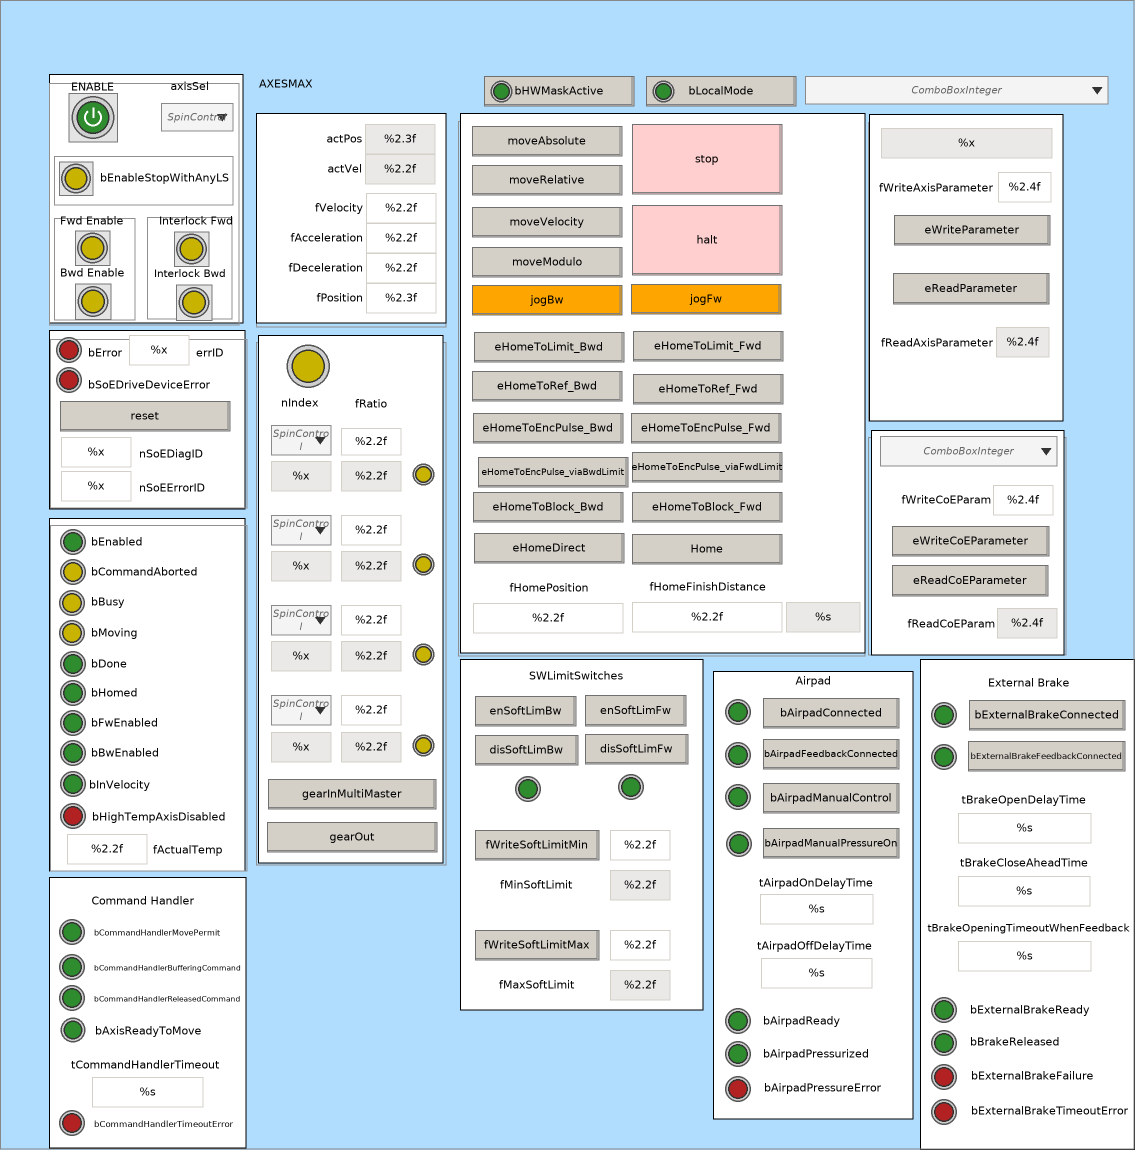
VISUALIZATION MainVisu  // 1135x1150
    Rectangle (49,518 196x353)
    Rectangle (49,330 196x179)
    Rectangle (49,877 197x271)
    Rectangle (49,74 194x249)
    GroupBox (868,114 195x307)
        Rectangle (1,0 194x307)
        Textfield (13,14 171x30), "%x", text variable: astAxes[MAIN.hmiAxisSelection].stConfig.eAxisParameters
            OnMouseClick: write GVL.astAxes[MAIN.hmiAxisSelection].stConfig.eAxisParameters via Default
        Textfield (130,58 53x30), "%2.4f", text variable: astAxes[MAIN.hmiAxisSelection].stConfig.fWriteAxisParameter
            OnMouseClick: write GVL.astAxes[MAIN.hmiAxisSelection].stConfig.fWriteAxisParameter via Default
        Button (26,101 156x30), "eWriteParameter", input disabled if: GVL.astAxes[MAIN.hmiAxisSelection].stStatus.bGeared, text list: "languageSupport", text index: "eWriteParameter"
            OnMouseClick: execute { GVL.astAxes[MAIN.hmiAxisSelection].stControl.eCommand:=E_MotionFunctions.eWriteParameter; GVL.astAxes[MAIN.hmiAxisSelection].stControl.bExecute:=TRUE; }
        Button (25,159 156x31), "eReadParameter", input disabled if: GVL.astAxes[MAIN.hmiAxisSelection].stStatus.bGeared, text list: 'languageSupport', text index: "eReadParameter"
            OnMouseClick: execute { GVL.astAxes[MAIN.hmiAxisSelection].stControl.eCommand:=E_MotionFunctions.eReadParameter; GVL.astAxes[MAIN.hmiAxisSelection].stControl.bExecute:=TRUE; }
        Textfield (128,213 53x30), "%2.4f", text variable: astAxes[MAIN.hmiAxisSelection].stConfig.fReadAxisParameter
            OnMouseClick: write GVL.astAxes[MAIN.hmiAxisSelection].stConfig.fReadAxisParameter via Default
    GroupBox (458,113 407x543)
        Rectangle (2,0 405x540)
        Button (174,92 150x70), "halt", pressed state: GVL.astAxes[Main.hmiAxisSelection].stControl.bHalt, input disabled if: GVL.astAxes[MAIN.hmiAxisSelection].stStatus.bGeared, text list: "languageSupport", text index: "halt"
            toggle GVL.astAxes[Main.hmiAxisSelection].stControl.bHalt
        Button (174,421 150x30), "Home", input disabled if: GVL.astAxes[MAIN.hmiAxisSelection].stStatus.bGeared, text list: 'languageSupport', text index: "Home"
            OnMouseClick: execute { GVL.astAxes[Main.hmiAxisSelection].stControl.eCommand:=E_MotionFunctions.eHome; GVL.astAxes[Main.hmiAxisSelection].stControl.bExecute:=TRUE; }
        Button (15,379 150x30), "eHomeToBlock_Bwd", input disabled if: GVL.astAxes[MAIN.hmiAxisSelection].stStatus.bGeared, text list: 'languageSupport', text index: "eHomeToBlock_Bwd"
            OnMouseClick: execute {
                GVL.astAxes[Main.hmiAxisSelection].stControl.eCommand:=E_MotionFunctions.eHome;
                GVL.astAxes[Main.hmiAxisSelection].stConfig.eHomeSeq:=E_HomingRoutines.eHomeToBlock_Bwd;
                GVL.astAxes[Main.hmiAxisSelection].stControl.bExecute:=TRUE;
            }
        Button (14,258 150x30), "eHomeToRef_Bwd", input disabled if: GVL.astAxes[MAIN.hmiAxisSelection].stStatus.bGeared, text list: 'languageSupport', text index: "eHomeToRef_Bwd"
            OnMouseClick: execute {
                GVL.astAxes[Main.hmiAxisSelection].stControl.eCommand:=E_MotionFunctions.eHome;
                GVL.astAxes[Main.hmiAxisSelection].stConfig.eHomeSeq:=E_HomingRoutines.eHomeToRef_Bwd;
                GVL.astAxes[Main.hmiAxisSelection].stControl.bExecute:=TRUE;
            }
        Button (14,13 150x30), "moveAbsolute", text list: "languageSupport", text index: "moveAbsolute"
            OnMouseClick: execute { GVL.astAxes[MAIN.hmiAxisSelection].stControl.eCommand:=E_MotionFunctions.eMoveAbsolute; GVL.astAxes[MAIN.hmiAxisSelection].stControl.bExecute:=TRUE; }
        Button (14,94 150x30), "moveVelocity", input disabled if: GVL.astAxes[MAIN.hmiAxisSelection].stStatus.bGeared, text list: "languageSupport", text index: "moveVelocity"
            OnMouseClick: execute { GVL.astAxes[Main.hmiAxisSelection].stControl.eCommand:=E_MotionFunctions.eMoveVelocity; GVL.astAxes[Main.hmiAxisSelection].stControl.bExecute:=TRUE; }
        Button (14,52 150x30), "moveRelative", input disabled if: GVL.astAxes[MAIN.hmiAxisSelection].stStatus.bGeared, text list: "languageSupport", text index: "moveRelative"
            OnMouseClick: execute { GVL.astAxes[Main.hmiAxisSelection].stControl.eCommand:=E_MotionFunctions.eMoveRelative; GVL.astAxes[Main.hmiAxisSelection].stControl.bExecute:=TRUE; }
        Button (14,134 150x30), "moveModulo", input disabled if: GVL.astAxes[MAIN.hmiAxisSelection].stStatus.bGeared, text list: "languageSupport", text index: "moveModulo"
            OnMouseClick: execute { GVL.astAxes[Main.hmiAxisSelection].stControl.eCommand:=E_MotionFunctions.eMoveModulo; GVL.astAxes[Main.hmiAxisSelection].stControl.bExecute:=TRUE; }
        Button (174,11 150x70), "stop", pressed state: GVL.astAxes[Main.hmiAxisSelection].stControl.bStop, input disabled if: GVL.astAxes[MAIN.hmiAxisSelection].stStatus.bGeared, text list: "languageSupport", text index: "stop"
            toggle GVL.astAxes[Main.hmiAxisSelection].stControl.bStop
        Button (14,172 150x30), "jogBw", text list: "languageSupport", text index: "jogBw"
            OnMouseDown: execute {
                GVL.astAxes[Main.hmiAxisSelection].stControl.eCommand:=E_MotionFunctions.eMoveVelocity;
                GVL.astAxes[Main.hmiAxisSelection].stControl.fVelocity:=-ABS(GVL.astAxes[Main.hmiAxisSelection].stControl.fJogVelocity);
                GVL.astAxes[Main.hmiAxisSelection].stControl.bExecute:= TRUE;
            }
            OnMouseUp: execute { GVL.astAxes[Main.hmiAxisSelection].stControl.bHalt:= TRUE; }
        Button (173,171 150x30), "jogFw", text list: "languageSupport", text index: "jogFw"
            OnMouseDown: execute {
                GVL.astAxes[Main.hmiAxisSelection].stControl.eCommand:=E_MotionFunctions.eMoveVelocity;
                GVL.astAxes[Main.hmiAxisSelection].stControl.fVelocity:=ABS(GVL.astAxes[Main.hmiAxisSelection].stControl.fJogVelocity);
                GVL.astAxes[Main.hmiAxisSelection].stControl.bExecute:= TRUE;
            }
            OnMouseUp: execute { GVL.astAxes[Main.hmiAxisSelection].stControl.bHalt:= TRUE; }
        Button (175,261 150x30), "eHomeToRef_Fwd", input disabled if: GVL.astAxes[MAIN.hmiAxisSelection].stStatus.bGeared, text list: "languageSupport", text index: "eHomeToRef_Fwd"
            OnMouseClick: execute {
                GVL.astAxes[Main.hmiAxisSelection].stControl.eCommand:=E_MotionFunctions.eHome;
                GVL.astAxes[Main.hmiAxisSelection].stConfig.eHomeSeq:=E_HomingRoutines.eHomeToRef_Fwd;
                GVL.astAxes[Main.hmiAxisSelection].stControl.bExecute:=TRUE;
            }
        Button (175,218 150x30), "eHomeToLimit_Fwd", input disabled if: GVL.astAxes[MAIN.hmiAxisSelection].stStatus.bGeared, text list: "languageSupport", text index: "eHomeToLimit_Fwd"
            OnMouseClick: execute {
                GVL.astAxes[Main.hmiAxisSelection].stControl.eCommand:=E_MotionFunctions.eHome;
                GVL.astAxes[Main.hmiAxisSelection].stConfig.eHomeSeq:=E_HomingRoutines.eHomeToLimit_Fwd;
                GVL.astAxes[Main.hmiAxisSelection].stControl.bExecute:=TRUE;
            }
        Button (16,219 150x30), "eHomeToLimit_Bwd", input disabled if: GVL.astAxes[MAIN.hmiAxisSelection].stStatus.bGeared, text list: 'languageSupport', text index: "eHomeToLimit_Bwd"
            OnMouseClick: execute {
                GVL.astAxes[Main.hmiAxisSelection].stControl.eCommand:=E_MotionFunctions.eHome;
                GVL.astAxes[Main.hmiAxisSelection].stConfig.eHomeSeq:=E_HomingRoutines.eHomeToLimit_Bwd;
                GVL.astAxes[Main.hmiAxisSelection].stControl.bExecute:=TRUE;
            }
        Button (15,300 150x30), "eHomeToEncPulse_Bwd", input disabled if: GVL.astAxes[MAIN.hmiAxisSelection].stStatus.bGeared, text list: 'languageSupport', text index: "eHomeToEncPulse_Bwd"
            OnMouseClick: execute {
                GVL.astAxes[Main.hmiAxisSelection].stControl.eCommand:=E_MotionFunctions.eHome;
                GVL.astAxes[Main.hmiAxisSelection].stConfig.eHomeSeq:=E_HomingRoutines.eHomeToEncPulse_Bwd;
                GVL.astAxes[Main.hmiAxisSelection].stControl.bExecute:=TRUE;
            }
        Button (173,300 150x30), "eHomeToEncPulse_Fwd", input disabled if: GVL.astAxes[MAIN.hmiAxisSelection].stStatus.bGeared, text list: "languageSupport", text index: "eHomeToEncPulse_Fwd"
            OnMouseClick: execute {
                GVL.astAxes[Main.hmiAxisSelection].stControl.eCommand:=E_MotionFunctions.eHome;
                GVL.astAxes[Main.hmiAxisSelection].stConfig.eHomeSeq:=E_HomingRoutines.eHomeToEncPulse_Fwd;
                GVL.astAxes[Main.hmiAxisSelection].stControl.bExecute:=TRUE;
            }
        Button (174,339 150x30), "eHomeToEncPulse_viaFwdLimit", input disabled if: GVL.astAxes[MAIN.hmiAxisSelection].stStatus.bGeared, text list: "languageSupport", text index: "eHomeToEncPulse_viaFwdLimit"
            OnMouseClick: execute {
                GVL.astAxes[Main.hmiAxisSelection].stControl.eCommand:=E_MotionFunctions.eHome;
                GVL.astAxes[Main.hmiAxisSelection].stConfig.eHomeSeq:=E_HomingRoutines.eHomeToEncPulse_viaFwdLimit;
                GVL.astAxes[Main.hmiAxisSelection].stControl.bExecute:=TRUE;
            }
        Button (20,344 150x30), "eHomeToEncPulse_viaBwdLimit", input disabled if: GVL.astAxes[MAIN.hmiAxisSelection].stStatus.bGeared, text list: 'languageSupport', text index: "eHomeToEncPulse_viaBwdLimit"
            OnMouseClick: execute {
                GVL.astAxes[Main.hmiAxisSelection].stControl.eCommand:=E_MotionFunctions.eHome;
                GVL.astAxes[Main.hmiAxisSelection].stConfig.eHomeSeq:=E_HomingRoutines.eHomeToEncPulse_viaBwdLimit;
                GVL.astAxes[Main.hmiAxisSelection].stControl.bExecute:=TRUE;
            }
        Button (174,379 150x30), "eHomeToBlock_Fwd", input disabled if: GVL.astAxes[MAIN.hmiAxisSelection].stStatus.bGeared, text list: "languageSupport", text index: "eHomeToBlock_Fwd"
            OnMouseClick: execute {
                GVL.astAxes[Main.hmiAxisSelection].stControl.eCommand:=E_MotionFunctions.eHome;
                GVL.astAxes[Main.hmiAxisSelection].stConfig.eHomeSeq:=E_HomingRoutines.eHomeToBlock_Fwd;
                GVL.astAxes[Main.hmiAxisSelection].stControl.bExecute:=TRUE;
            }
        Button (16,420 150x30), "eHomeDirect", input disabled if: GVL.astAxes[MAIN.hmiAxisSelection].stStatus.bGeared, text list: 'languageSupport', text index: "eHomeDirect"
            OnMouseClick: execute {
                GVL.astAxes[Main.hmiAxisSelection].stControl.eCommand:=E_MotionFunctions.eHome;
                GVL.astAxes[Main.hmiAxisSelection].stConfig.eHomeSeq:=E_HomingRoutines.eHomeDirect;
                GVL.astAxes[Main.hmiAxisSelection].stControl.bExecute:=TRUE;
            }
        Textfield (15,490 150x30), "%2.2f", text variable: GVL.astAxes[MAIN.hmiAxisSelection].stConfig.fHomePosition
            OnMouseClick: write the text variable via Default
        Textfield (174,489 150x30), "%2.2f", text variable: GVL.astAxes[MAIN.hmiAxisSelection].stConfig.fHomeFinishDistance, text list: ''
            OnMouseClick: write the text variable via Default
        Textfield (175,459 150x30), "fHomeFinishDistance", text list: "languageSupport", text index: "fHomeFinishDistance"
        Textfield (16,460 150x30), "fHomePosition", text list: "languageSupport", text index: "fHomePosition"
        Textfield (328,489 74x30), "%s", text variable: SEL(GVL.astAxes[Main.hmiAxisSelection].stConfig.stHomingConfig.bAbsoluteMoveAtFinishHoming, 'Relative', 'Absolute');
    GroupBox (256,334 190x531)
        Rectangle (2,1 185x528)
        SpinControl (15,91 60x30), variable: GVL.astAxes[MAIN.hmiAxisSelection].stConfig.astMultiMasterAxis[1].nIndex
            p651134158: GVL_APP.nAXIS_NUM
        Textfield (85,94 60x27), "%2.2f", text variable: GVL.astAxes[MAIN.hmiAxisSelection].stConfig.astMultiMasterAxis[1].fRatio
            OnMouseClick: write the text variable via Default
        Textfield (80,55 70x30), "fRatio", text list: "languageSupport", text index: "gearRatio"
        Button (12,445 168x30), "gearInMultiMaster", text list: "languageSupport", text index: "gearIn"
            OnMouseClick: execute { GVL.astAxes[Main.hmiAxisSelection].stControl.eCommand:=E_MotionFunctions.eGearInMultiMaster; GVL.astAxes[Main.hmiAxisSelection].stControl.bExecute:=TRUE; }
        SpinControl (15,181 60x30), variable: GVL.astAxes[MAIN.hmiAxisSelection].stConfig.astMultiMasterAxis[2].nIndex
            p651134158: GVL_APP.nAXIS_NUM
        SpinControl (15,271 60x30), variable: GVL.astAxes[MAIN.hmiAxisSelection].stConfig.astMultiMasterAxis[3].nIndex
            p651134158: GVL_APP.nAXIS_NUM
        SpinControl (15,361 60x30), variable: GVL.astAxes[MAIN.hmiAxisSelection].stConfig.astMultiMasterAxis[4].nIndex
            p651134158: GVL_APP.nAXIS_NUM
        Textfield (85,181 60x30), "%2.2f", text variable: GVL.astAxes[MAIN.hmiAxisSelection].stConfig.astMultiMasterAxis[2].fRatio
            OnMouseClick: write the text variable via Default
        Textfield (85,271 60x30), "%2.2f", text variable: GVL.astAxes[MAIN.hmiAxisSelection].stConfig.astMultiMasterAxis[3].fRatio
            OnMouseClick: write the text variable via Default
        Textfield (85,361 60x30), "%2.2f", text variable: GVL.astAxes[MAIN.hmiAxisSelection].stConfig.astMultiMasterAxis[4].fRatio
            OnMouseClick: write the text variable via Default
        Button (11,488 170x30), "gearOut", text list: "languageSupport", text index: "gearOut"
            OnMouseClick: execute { GVL.astAxes[Main.hmiAxisSelection].stControl.eCommand:=E_MotionFunctions.eGearOut; GVL.astAxes[Main.hmiAxisSelection].stControl.bExecute:=TRUE; }
        Textfield (9,54 70x30), "nIndex", text list: "languageSupport", text index: "masterGear"
        Textfield (85,127 60x30), "%2.2f", text variable: GVL.astAxes[MAIN.hmiAxisSelection].Axis.PlcToNc.GearRatio1
        Textfield (15,127 60x30), "%x", text variable: GVL.astAxes[MAIN.hmiAxisSelection].stConfig.astMultiMasterAxisLatched[1].nIndex
        Textfield (85,217 60x30), "%2.2f", text variable: GVL.astAxes[MAIN.hmiAxisSelection].Axis.PlcToNc.GearRatio2
        Textfield (15,217 60x30), "%x", text variable: GVL.astAxes[MAIN.hmiAxisSelection].stConfig.astMultiMasterAxisLatched[2].nIndex
        Textfield (85,307 60x30), "%2.2f", text variable: GVL.astAxes[MAIN.hmiAxisSelection].Axis.PlcToNc.GearRatio3
        Textfield (15,307 60x30), "%x", text variable: GVL.astAxes[MAIN.hmiAxisSelection].stConfig.astMultiMasterAxisLatched[3].nIndex
        Textfield (85,398 60x30), "%2.2f", text variable: GVL.astAxes[MAIN.hmiAxisSelection].Axis.PlcToNc.GearRatio4
        Textfield (15,398 60x30), "%x", text variable: GVL.astAxes[MAIN.hmiAxisSelection].stConfig.astMultiMasterAxisLatched[4].nIndex
        Lamp1 (155,399 25x25), variable: GVL.astAxes[MAIN.hmiAxisSelection].stStatus.bCoupledGear4, style: Lamp-Lamp1-Yellow
        Lamp1 (155,308 25x25), variable: GVL.astAxes[MAIN.hmiAxisSelection].stStatus.bCoupledGear3, style: Lamp-Lamp1-Yellow
        Lamp1 (155,218 25x25), variable: GVL.astAxes[MAIN.hmiAxisSelection].stStatus.bCoupledGear2, style: Lamp-Lamp1-Yellow
        Lamp1 (155,128 25x25), variable: GVL.astAxes[MAIN.hmiAxisSelection].stStatus.bCoupledGear1, style: Lamp-Lamp1-Yellow
        Lamp1 (27,7 50x50), variable: GVL.astAxes[MAIN.hmiAxisSelection].stStatus.bGeared, style: Lamp-Lamp1-Yellow
    Textfield (256,69 196x30), "AXESMAX", text variable: GVL_APP.nAXIS_NUM, text list: "languageSupport", text index: "axesAvailable"
    GroupBox (50,517 197x354)
        Lamp1 (8,10 30x30), variable: GVL.astAxes[MAIN.hmiAxisSelection].stStatus.bEnabled, style: Lamp-Lamp1-Green
        Textfield (38,10 140x30), "bEnabled", text list: "languageSupport", text index: "bEnabled"
        Lamp1 (8,40 30x30), variable: GVL.astAxes[MAIN.hmiAxisSelection].stStatus.bCommandAborted, style: Lamp-Lamp1-Yellow
        Textfield (38,40 140x30), "bCommandAborted", text list: "languageSupport", text index: "bCommandAborted"
        Textfield (38,70 140x30), "bBusy", text list: "languageSupport", text index: "bBusy"
        Lamp1 (8,132 30x30), variable: GVL.astAxes[MAIN.hmiAxisSelection].stStatus.bDone, style: Lamp-Lamp1-Green
        Textfield (38,132 140x30), "bDone", text list: 'languageSupport', text index: "bDone"
        Lamp1 (8,161 30x30), variable: GVL.astAxes[MAIN.hmiAxisSelection].stStatus.bHomed, style: Lamp-Lamp1-Green
        Textfield (38,161 140x30), "bHomed", text list: "languageSupport", text index: "bHomed"
        Lamp1 (8,191 30x30), variable: GVL.astAxes[MAIN.hmiAxisSelection].stStatus.bFwEnabled, style: Lamp-Lamp1-Green
        Lamp1 (8,221 30x30), variable: GVL.astAxes[MAIN.hmiAxisSelection].stStatus.bBwEnabled, style: Lamp-Lamp1-Green
        Textfield (38,191 140x30), "bFwEnabled", text list: "languageSupport", text index: "bFwEnabled"
        Textfield (38,221 140x30), "bBwEnabled", text list: "languageSupport", text index: "bBwEnabled"
        Lamp1 (7,71 30x30), variable: GVL.astAxes[MAIN.hmiAxisSelection].stStatus.bBusy, style: Lamp-Lamp1-Yellow
        Lamp1 (8,252 30x30), variable: GVL.astAxes[MAIN.hmiAxisSelection].stStatus.bInVelocity, style: Lamp-Lamp1-Green
        Lamp1 (8,284 30x30), variable: GVL.astAxes[MAIN.hmiAxisSelection].stStatus.bHighTempAxisDisabled, style: Lamp-Lamp1-Red
        Textfield (17,317 80x30), "%2.2f", text variable: GVL.astAxes[MAIN.hmiAxisSelection].stStatus.fActTemperature
        Textfield (100,318 79x30), "fActualTemp", text list: "languageSupport", text index: "fActualTemp"
        Textfield (36,253 140x30), "bInVelocity", text list: 'languageSupport', text index: "bInVelocity"
        Textfield (39,285 140x30), "bHighTempAxisDisabled", text list: 'languageSupport', text index: "bHighTempDisable"
        Lamp1 (7,101 30x30), variable: GVL.astAxes[MAIN.hmiAxisSelection].stStatus.bMoving, style: Lamp-Lamp1-Yellow
        Textfield (38,101 140x30), "bMoving", text list: "languageSupport", text index: "bMoving"
    GroupBox (256,113 190x214)
        Rectangle (0,0 190x210)
        Textfield (10,80 100x30), "fVelocity", text list: "languageSupport", text index: "fVelocity"
        Textfield (110,80 70x30), "%2.2f", text variable: GVL.astAxes[MAIN.hmiAxisSelection].stControl.fVelocity
            OnMouseClick: write the text variable via Default
        Textfield (10,110 100x30), "fAcceleration", text list: "languageSupport", text index: "fAcceleration"
        Textfield (110,110 70x30), "%2.2f", text variable: GVL.astAxes[MAIN.hmiAxisSelection].stControl.fAcceleration
            OnMouseClick: write the text variable via Default
        Textfield (10,140 100x30), "fDeceleration", text list: "languageSupport", text index: "fDeceleration"
        Textfield (110,140 70x30), "%2.2f", text variable: GVL.astAxes[MAIN.hmiAxisSelection].stControl.fDeceleration
            OnMouseClick: write the text variable via Default
        Textfield (10,170 100x30), "fPosition", text list: "languageSupport", text index: "fPosition"
        Textfield (110,170 70x30), "%2.3f", text variable: GVL.astAxes[MAIN.hmiAxisSelection].stControl.fPosition
            OnMouseClick: write the text variable via Default
        Textfield (109,11 70x30), "%2.3f", text variable: GVL.astAxes[MAIN.hmiAxisSelection].stStatus.fActPosition
        Textfield (9,11 100x30), "actPos", text list: "languageSupport", text index: "actposition"
        Textfield (9,41 100x30), "actVel", text list: "languageSupport", text index: "actVelocity"
        Textfield (109,41 70x30), "%2.2f", text variable: GVL.astAxes[MAIN.hmiAxisSelection].stStatus.fActVelocity
    Group (646,76 149x30), text variable: GVL.bLocalMode
        Button (0,0 150x30), "bLocalMode", text list: 'languageSupport', text index: 'bLocalMode'
            OnMouseClick: toggle GVL.bLocalMode
        Lamp1 (5,3 25x25), variable: GVL.bLocalMode, style: Lamp-Lamp1-Green
    ComboBoxInteger (805,76 303x28), variable: GVL.astAxes[MAIN.hmiAxisSelection].stConfig.eAxisParameters, text list: 'ParameterTextList'
    Group (484,76 148x30), text variable: GVL.astAxes[MAIN.hmiAxisSelection].stControl.bHWMaskActive
        Button (0,0 150x30), "bHWMaskActive", text list: 'languageSupport', text index: 'bHWMaskActive'
            OnMouseClick: toggle GVL.astAxes[MAIN.hmiAxisSelection].stControl.bHWMaskActive
        Lamp1 (5,3 25x25), variable: GVL.astAxes[MAIN.hmiAxisSelection].stControl.bHWMaskActive, style: Lamp-Lamp1-Green
    Textfield (855,328 141x30), "fReadAxisParameter", text list: "languageSupport", text index: "fReadAxisParameter"
    Textfield (855,173 141x30), "fWriteAxisParameter", text list: "languageSupport", text index: "fWriteAxisParameter"
    Group (49,75 197x250)
        GroupBox (0,0 190x250)
            GroupBox (98,134 85x110)
                PushSwitchLed (27,19 35x42), variable: astAxes[MAIN.hmiAxisSelection].stControl.bInterlockFwd, behaviour: TOGGLE, style: Switch-PushSwitchLed-Yellow
                Textfield (4,51 76x27), "Interlock Bwd", text list: 'languageSupport', text index: "bAxisInterlockBwd"
            Textfield (107,133 76x26), "Interlock Fwd", text list: 'languageSupport', text index: "bAxisInterlockFwd"
            GroupBox (5,135 81x110)
                Textfield (3,50 76x26), "Bwd Enable", text list: 'languageSupport', text index: "enBW"
                Textfield (3,-2 76x26), "Fwd Enable", text list: 'languageSupport', text index: "enFW"
            PushSwitchLed (127,208 36x39), variable: GVL.astAxes[MAIN.hmiAxisSelection].stControl.bInterlockBwd, behaviour: TOGGLE, style: Switch-PushSwitchLed-Yellow
            PushSwitchLed (26,152 35x42), variable: GVL.astAxes[MAIN.hmiAxisSelection].stInputs.bLimitFwd, behaviour: TOGGLE, style: Switch-PushSwitchLed-Yellow
            PushSwitchLed (26,207 36x39), variable: GVL.astAxes[MAIN.hmiAxisSelection].stInputs.bLimitBwd, behaviour: TOGGLE, style: Switch-PushSwitchLed-Yellow
            PowerSwitch (19,18 50x49), variable: GVL.astAxes[MAIN.hmiAxisSelection].stControl.bEnable, behaviour: TOGGLE, style: Switch-PowerSwitch-Green
            SpinControl (112,28 72x28), variable: MAIN.hmiAxisSelection
                p651134158: GVL_APP.nAXIS_NUM
            GroupBox (5,73 179x57)
                PushSwitchLed (5,13 34x35), variable: astAxes[MAIN.hmiAxisSelection].stConfig.bEnableStopWithAnyLimitSwitch, behaviour: TOGGLE, style: Switch-PushSwitchLed-Yellow
            Textfield (99,0 84x23), "axisSel", text variable: GVL_APP.nAXIS_NUM, text list: "languageSupport", text index: "axisSel"
        Textfield (19,0 62x24), "ENABLE", text list: 'languageSupport', text index: "enable"
        Textfield (48,90 135x26), "bEnableStopWithAnyLS", text list: 'languageSupport', text index: "bEnableStopWithAnyLimitSwitch"
    GroupBox (868,429 198x226)
        Rectangle (3,1 193x225)
        Textfield (6,56 120x30), "fWriteCoEParam", text list: "languageSupport", text index: "fWriteCoEParameter"
        Textfield (125,56 60x30), "%2.4f", text variable: astAxes[MAIN.hmiAxisSelection].stConfig.stCoEParameters.aParWrite[1]
            OnMouseClick: write GVL.astAxes[MAIN.hmiAxisSelection].stConfig.stCoEParameters.aParWrite[1] via Default
        Button (24,97 157x30), "eWriteCoEParameter", text list: "languageSupport", text index: "eWriteCoEParameter"
            OnMouseClick: execute { GVL.astAxes[MAIN.hmiAxisSelection].stControl.eCommand:=E_MotionFunctions.eWriteCoEParameters; GVL.astAxes[MAIN.hmiAxisSelection].stControl.bExecute:=TRUE; }
        Button (24,136 156x31), "eReadCoEParameter", text list: 'languageSupport', text index: "eReadCoEParameter"
            OnMouseClick: execute { GVL.astAxes[MAIN.hmiAxisSelection].stControl.eCommand:=E_MotionFunctions.eReadCoEParameters; GVL.astAxes[MAIN.hmiAxisSelection].stControl.bExecute:=TRUE; }
        Textfield (10,180 120x30), "fReadCoEParam", text list: "languageSupport", text index: "fReadCoEParameter"
        Textfield (129,179 60x30), "%2.4f", text variable: astAxes[MAIN.hmiAxisSelection].stConfig.stCoEParameters.aParRead[1]
            OnMouseClick: write GVL.astAxes[MAIN.hmiAxisSelection].stConfig.stCoEParameters.aParRead[1] via Default
    ComboBoxInteger (880,436 177x30), variable: GVL.astAxes[MAIN.hmiAxisSelection].stConfig.stCoEParameters.eCoEParameters, text list: 'CoEParamTextList'
    Rectangle (460,659 243x351)
    Button (585,695 101x31), "enSoftLimFw", text list: "languageSupport", text index: "enSoftLimFw"
        OnMouseClick: execute {
            GVL.astAxes[Main.hmiAxisSelection].stConfig.eAxisParameters := E_AxisParameters.EnableLimitForward;
            GVL.astAxes[Main.hmiAxisSelection].stConfig.fWriteAxisParameter := 1.0;
            GVL.astAxes[Main.hmiAxisSelection].stControl.eCommand := E_MotionFunctions.eWriteParameter;
            GVL.astAxes[Main.hmiAxisSelection].stControl.bExecute := TRUE;
        }
    Button (585,734 103x30), "disSoftLimFw", text list: "languageSupport", text index: "disSoftLimFw"
        OnMouseClick: execute {
            GVL.astAxes[Main.hmiAxisSelection].stConfig.eAxisParameters := E_AxisParameters.EnableLimitForward;
            GVL.astAxes[Main.hmiAxisSelection].stConfig.fWriteAxisParameter := 0.0;
            GVL.astAxes[Main.hmiAxisSelection].stControl.eCommand := E_MotionFunctions.eWriteParameter;
            GVL.astAxes[Main.hmiAxisSelection].stControl.bExecute := TRUE;
        }
    Lamp1 (513,774 30x30), variable: GVL.astAxes[Main.hmiAxisSelection].stConfig.bEnMinSoftPosLimit, style: Lamp-Lamp1-Green
    Lamp1 (616,772 30x30), variable: GVL.astAxes[Main.hmiAxisSelection].stConfig.bEnMaxSoftPosLimit, style: Lamp-Lamp1-Green
    Button (475,696 101x30), "enSoftLimBw", text list: "languageSupport", text index: "enSoftLimBw"
        OnMouseClick: execute {
            GVL.astAxes[Main.hmiAxisSelection].stConfig.eAxisParameters := E_AxisParameters.EnableLimitBackward;
            GVL.astAxes[Main.hmiAxisSelection].stConfig.fWriteAxisParameter := 1.0;
            GVL.astAxes[Main.hmiAxisSelection].stControl.eCommand := E_MotionFunctions.eWriteParameter;
            GVL.astAxes[Main.hmiAxisSelection].stControl.bExecute := TRUE;
        }
    Textfield (501,661 150x30), "SWLimitSwitches", text list: "languageSupport", text index: "SWLimitSwitches"
    Button (475,735 103x30), "disSoftLimBw", text list: "languageSupport", text index: "disSoftLimBw"
        OnMouseClick: execute {
            GVL.astAxes[Main.hmiAxisSelection].stConfig.eAxisParameters := E_AxisParameters.EnableLimitBackward;
            GVL.astAxes[Main.hmiAxisSelection].stConfig.fWriteAxisParameter := 0.0;
            GVL.astAxes[Main.hmiAxisSelection].stControl.eCommand := E_MotionFunctions.eWriteParameter;
            GVL.astAxes[Main.hmiAxisSelection].stControl.bExecute := TRUE;
        }
    Rectangle (713,671 200x448)
    Lamp1 (723,697 30x30), variable: GVL.astAxes[MAIN.hmiAxisSelection].stConfig.stAirpadBrake.bAirpadConnected, style: Lamp-Lamp1-Green
    Button (763,739 136x30), "bAirpadFeedbackConnected", text list: "languageSupport", text index: "bAirpadFeedbackConnected"
        OnMouseClick: toggle GVL.astAxes[MAIN.hmiAxisSelection].stConfig.stAirpadBrake.bAirpadFeedbackConnected
    Lamp1 (723,740 30x30), variable: GVL.astAxes[MAIN.hmiAxisSelection].stConfig.stAirpadBrake.bAirpadFeedbackConnected, style: Lamp-Lamp1-Green
    Rectangle (920,659 215x491)
    Lamp1 (929,700 30x30), variable: GVL.astAxes[MAIN.hmiAxisSelection].stConfig.stAirpadBrake.bExternalBrakeConnected, style: Lamp-Lamp1-Green
    Button (969,700 156x30), "bExternalBrakeConnected", text list: "languageSupport", text index: "bExternalBrakeConnected"
        OnMouseClick: toggle GVL.astAxes[MAIN.hmiAxisSelection].stConfig.stAirpadBrake.bExternalBrakeConnected
    Textfield (760,1039 141x30), "bAirpadPressurized", text list: "languageSupport", text index: "bAirpadPressurized"
    Button (968,741 157x30), "bExternalBrakeFeedbackConnected", text list: "languageSupport", text index: "bExternalBrakeFeedbackConnected"
        OnMouseClick: toggle GVL.astAxes[MAIN.hmiAxisSelection].stConfig.stAirpadBrake.bExternalBrakeFeedbackConnected
    Lamp1 (929,742 30x30), variable: GVL.astAxes[MAIN.hmiAxisSelection].stConfig.stAirpadBrake.bExternalBrakeFeedbackConnected, style: Lamp-Lamp1-Green
    Textfield (967,1027 131x30), "bBrakeReleased", text list: 'languageSupport', text index: "bBrakeReleased"
    Textfield (760,894 113x30), "%s", text variable: GVL.astAxes[MAIN.hmiAxisSelection].stConfig.stAirpadBrake.tAirpadOnDelayTime
        OnMouseClick: write the text variable via Default
    Textfield (718,868 196x30), "tAirpadOnDelayTime", text list: "languageSupport", text index: "tAirpadOnDelayTime"
    Textfield (941,785 166x30), "tBrakeOpenDelayTime", text list: "languageSupport", text index: "tBrakeOpenDelayTime"
    Textfield (958,813 133x30), "%s", text variable: GVL.astAxes[MAIN.hmiAxisSelection].stConfig.stAirpadBrake.tBrakeOpenDelayTime
        OnMouseClick: write GVL.astAxes[MAIN.hmiAxisSelection].stConfig.stAirpadBrake.tBrakeOpenDelayTime via Default
    Textfield (941,848 166x30), "tBrakeCloseAheadTime", text list: "languageSupport", text index: "tBrakeCloseAheadTime"
    Textfield (958,876 132x30), "%s", text variable: GVL.astAxes[MAIN.hmiAxisSelection].stConfig.stAirpadBrake.tBrakeCloseAheadTime
        OnMouseClick: write the text variable via Default
    Lamp1 (929,1028 30x30), variable: GVL.astAxes[MAIN.hmiAxisSelection].stInputs.bBrakeReleased, style: Lamp-Lamp1-Green
    Lamp1 (723,1039 30x30), variable: GVL.astAxes[MAIN.hmiAxisSelection].stInputs.bAirpadPressurized, style: Lamp-Lamp1-Green
    Lamp1 (58,1016 30x28), variable: GVL.astAxes[MAIN.hmiAxisSelection].stStatus.bAxisReadyToMove, style: Lamp-Lamp1-Green
    Button (763,698 136x30), "bAirpadConnected", text list: 'languageSupport', text index: "bAirpadConnected"
        OnMouseClick: toggle GVL.astAxes[MAIN.hmiAxisSelection].stConfig.stAirpadBrake.bAirpadConnected
    Textfield (92,1016 137x30), "bAxisReadyToMove", text list: "languageSupport", text index: "bAxisReadyToMove"
    Textfield (91,953 150x30), "bCommandHandlerBufferingCommand", text list: "languageSupport", text index: "bCommandHandlerBufferingCommand"
    Lamp1 (57,952 30x30), variable: GVL.astAxes[MAIN.hmiAxisSelection].stStatus.bCommandHandlerBufferingCommand, style: Lamp-Lamp1-Green
    Lamp1 (723,1074 30x30), variable: GVL.astAxes[MAIN.hmiAxisSelection].stStatus.bAirpadPressureError, style: Lamp-Lamp1-Red
    Textfield (761,1073 129x30), "bAirpadPressureError", text list: "languageSupport", text index: "bAirpadPressureError"
    Textfield (958,941 133x30), "%s", text variable: GVL.astAxes[MAIN.hmiAxisSelection].stConfig.stAirpadBrake.tBrakeOpeningTimeoutWhenFeedback
        OnMouseClick: write the text variable via Default
    Textfield (922,913 213x30), "tBrakeOpeningTimeoutWhenFeedback", text list: "languageSupport", text index: "tBrakeOpeningTimeoutWhenFeedback"
    Lamp1 (929,1062 30x30), variable: GVL.astAxes[MAIN.hmiAxisSelection].stStatus.bExternalBrakeFailure, style: Lamp-Lamp1-Red
    Textfield (968,1061 145x30), "bExternalBrakeFailure", text list: "languageSupport", text index: "bExternalBrakeFailure"
    Lamp1 (929,1097 30x30), variable: GVL.astAxes[MAIN.hmiAxisSelection].stStatus.bExternalBrakeTimeoutError, style: Lamp-Lamp1-Red
    Textfield (968,1096 161x30), "bExternalBrakeTimeoutError", text list: "languageSupport", text index: "bExternalBrakeTimeoutError"
    Lamp1 (723,782 30x30), variable: GVL.astAxes[MAIN.hmiAxisSelection].stConfig.bAirpadManualControl, style: Lamp-Lamp1-Green
    Button (763,828 136x30), "bAirpadManualPressureOn", text list: "languageSupport", text index: "bAirpadManualPressureOn"
        OnMouseClick: toggle GVL.astAxes[MAIN.hmiAxisSelection].stControl.bAirpadManualPressureOn
    Lamp1 (724,829 30x30), variable: GVL.astAxes[MAIN.hmiAxisSelection].stControl.bAirpadManualPressureOn, style: Lamp-Lamp1-Green
    Button (763,783 136x30), "bAirpadManualControl", text list: "languageSupport", text index: "bAirpadManualControl"
        OnMouseClick: toggle GVL.astAxes[MAIN.hmiAxisSelection].stConfig.bAirpadManualControl
    Textfield (91,1109 138x30), "bCommandHandlerTimeoutError", text list: "languageSupport", text index: "bCommandHandlerTimeoutError"
    Lamp1 (57,1108 30x30), variable: GVL.astAxes[MAIN.hmiAxisSelection].stStatus.bCommandHandlerTimeoutError, style: Lamp-Lamp1-Red
    Textfield (68,886 150x30), "Command Handler", text list: 'languageSupport', text index: "CommandHandler"
    Textfield (930,668 198x30), "External Brake", text list: 'languageSupport', text index: "ExternalBrake"
    Textfield (719,666 189x30), "Airpad", text list: "languageSupport", text index: "Airpad"
    Textfield (760,1006 88x30), "bAirpadReady", text list: "languageSupport", text index: "bAirpadReady"
    Textfield (967,995 140x30), "bExternalBrakeReady", text list: "languageSupport", text index: "bExternalBrakeReady"
    Lamp1 (929,995 30x30), variable: GVL.astAxes[MAIN.hmiAxisSelection].stStatus.bExternalBrakeReady, style: Lamp-Lamp1-Green
    Lamp1 (723,1006 30x30), variable: GVL.astAxes[MAIN.hmiAxisSelection].stStatus.bAirpadReady, style: Lamp-Lamp1-Green
    Textfield (58,1050 175x30), "tCommandHandlerTimeout", text list: "languageSupport", text index: "tCommandHandlerTimeout"
    Textfield (92,1077 111x30), "%s", text variable: GVL.astAxes[MAIN.hmiAxisSelection].stConfig.tCommandHandlerTimeout
        OnMouseClick: write the text variable via Default
    Textfield (91,918 133x30), "bCommandHandlerMovePermit", text list: "languageSupport", text index: "bCommandHandlerMovePermit"
    Lamp1 (57,917 30x30), variable: GVL.astAxes[MAIN.hmiAxisSelection].stStatus.bCommandHandlerMovePermit, style: Lamp-Lamp1-Green
    Textfield (727,931 175x30), "tAirpadOffDelayTime", text list: "languageSupport", text index: "tAirpadOffDelayTime"
    Textfield (761,958 111x30), "%s", text variable: GVL.astAxes[MAIN.hmiAxisSelection].stConfig.stAirpadBrake.tAirpadOffDelayTime
        OnMouseClick: write the text variable via Default
    GroupBox (50,331 197x177)
        Lamp1 (4,4 30x30), variable: GVL.astAxes[MAIN.hmiAxisSelection].stStatus.bError, style: Lamp-Lamp1-Red
        Textfield (35,7 37x30), "bError", text list: "languageSupport", text index: "bError"
        Button (10,70 170x30), "reset", pressed state: GVL.astAxes[Main.hmiAxisSelection].stControl.bReset, text list: "languageSupport", text index: "reset"
            OnMouseClick: toggle GVL.astAxes[Main.hmiAxisSelection].stControl.bReset
        Lamp1 (4,34 30x30), variable: GVL.astAxes[MAIN.hmiAxisSelection].stStatus.bSoEDriveDeviceError, style: Lamp-Lamp1-Red
        Textfield (11,106 70x30), "%x", text variable: GVL.astAxes[MAIN.hmiAxisSelection].stStatus.nSoEDiagID
        Textfield (11,140 70x30), "%x", text variable: GVL.astAxes[MAIN.hmiAxisSelection].stStatus.nSoEErrorID
    Textfield (85,370 134x30), "bSoEDriveDeviceError", text list: "languageSupport", text index: "bSoEDriveDeviceError"
    Textfield (136,439 100x30), "nSoEDiagID", text list: "languageSupport", text index: "nSoEDiagID"
    Textfield (136,473 100x30), "nSoEErrorID", text list: "languageSupport", text index: "nSoEErrorID"
    Textfield (129,335 60x30), "%x", text variable: GVL.astAxes[MAIN.hmiAxisSelection].stStatus.nErrorID
    Textfield (193,338 48x30), "errID", text list: "languageSupport", text index: "errID"
    Textfield (610,830 60x30), "%2.2f", text variable: GVL.astAxes[MAIN.hmiAxisSelection].stConfig.fWriteMinSoftLimit
        OnMouseClick: write GVL.astAxes[MAIN.hmiAxisSelection].stConfig.fWriteMinSoftLimit via Default
    Button (475,830 124x30), "fWriteSoftLimitMin", text list: "languageSupport", text index: "fWriteSoftLimitMin"
        OnMouseClick: execute {
            GVL.astAxes[Main.hmiAxisSelection].stConfig.eAxisParameters := E_AxisParameters.SWLimitBackward;
            GVL.astAxes[Main.hmiAxisSelection].stConfig.fWriteAxisParameter := GVL.astAxes[MAIN.hmiAxisSelection].stConfig.fWriteMinSoftLimit;
            GVL.astAxes[Main.hmiAxisSelection].stControl.eCommand := E_MotionFunctions.eWriteParameter;
            GVL.astAxes[Main.hmiAxisSelection].stControl.bExecute := TRUE;
        }
    Textfield (475,870 123x30), "fMinSoftLimit", text list: "languageSupport", text index: "fMinSoftLimit"
    Textfield (610,930 60x30), "%2.2f", text variable: GVL.astAxes[MAIN.hmiAxisSelection].stConfig.fWriteMaxSoftLimit
        OnMouseClick: write GVL.astAxes[MAIN.hmiAxisSelection].stConfig.fWriteMaxSoftLimit via Edit
    Button (475,930 124x30), "fWriteSoftLimitMax", text list: "languageSupport", text index: "fWriteSoftLimitMax"
        OnMouseClick: execute {
            GVL.astAxes[Main.hmiAxisSelection].stConfig.eAxisParameters := E_AxisParameters.SWLimitForward;
            GVL.astAxes[Main.hmiAxisSelection].stConfig.fWriteAxisParameter := GVL.astAxes[MAIN.hmiAxisSelection].stConfig.fWriteMaxSoftLimit;
            GVL.astAxes[Main.hmiAxisSelection].stControl.eCommand := E_MotionFunctions.eWriteParameter;
            GVL.astAxes[Main.hmiAxisSelection].stControl.bExecute := TRUE;
        }
    Textfield (475,970 124x30), "fMaxSoftLimit", text list: "languageSupport", text index: "fMaxSoftLimit"
    Textfield (610,870 60x30), "%2.2f", text variable: GVL.astAxes[Main.hmiAxisSelection].stConfig.fMinSoftPosLimit
    Textfield (610,970 60x30), "%2.2f", text variable: GVL.astAxes[Main.hmiAxisSelection].stConfig.fMaxSoftPosLimit
    Lamp1 (57,983 30x30), variable: GVL.astAxes[MAIN.hmiAxisSelection].stStatus.bCommandHandlerReleasedMoveCmd, style: Lamp-Lamp1-Green
    Textfield (91,984 150x30), "bCommandHandlerReleasedCommand", text list: "languageSupport", text index: "bCommandHandlerReleasedCommand"
    hotkey HotkeyInput Id=481037385728, Key=KeyDown=True, KeyName=RETURN_KEY, VisuElemId=753
    hotkey HotkeyInput Id=481038434304, Key=KeyName=RETURN_KEY, VisuElemId=753
END_VISUALIZATION

(* stored: Version 1.1.0.1
   Visu MainVisu: Id {98c8ae72-e756-4d11-b6a5-5914882e2424} *)
